// TwinCAT 3 PLC project PLCSim
// ProgramVersion: 3.1.4022.3
// libraries:
//   Tc2_Standard, * (Beckhoff Automation GmbH)
//   Tc2_System, * (Beckhoff Automation GmbH)
//   Tc3_Module, * (Beckhoff Automation GmbH)
//   VisuSymbols,3.5.10.0,System
// project tree:
//   / GlobalTextList.TcGTLO, PlcTask.TcTTO (not stored), Visualization Manager.TcVMO (not stored)
//   POUs/ MAIN.TcPOU
//   VISUs/ Visualization.TcVIS

// ---- POUs/MAIN.TcPOU
PROGRAM MAIN
VAR
	ixLampStarted	AT %I* : BOOL;
	ixSliderAout 	AT %I* : BOOL; 
	ixSliderAin 	AT %I* : BOOL; 
	ixSliderBout 	AT %I* : BOOL; 
	ixSliderBin 	AT %I* : BOOL; 
	ixDrillDown 	AT %I* : BOOL;
	ixDrillUp		AT %I* : BOOL;
	
	qxButtonStart	AT %Q* : BOOL;
	qxButtonStop	AT %Q* : BOOL;
	qxSliderAout	AT %Q* : BOOL;
	qxSliderAin		AT %Q* : BOOL;
	qxSliderBout	AT %Q* : BOOL;
	qxSliderBin		AT %Q* : BOOL;
	qxDrillUp		AT %Q* : BOOL;
	qxDrillDown		AT %Q* : BOOL;
	
	mxReset 		: BOOL;
	mxCubeInvisible : BOOL;
	
	
	nPosSliderA 	: INT:=0;
	nPosSliderB 	: INT:=0;
	nPosDrill 		: INT:=0;
	nPosXCube		: INT:=0;
	nPosYCube		: INT:=0;
	nSpeed 			: INT:=1;
	nCnt			: INT:=0;
	nErrorCnt		: INT:=0;
	nSeq: INT;
	
	fbTONAin:TON;
	fbTONAout:TON;
	fbTONBin:TON;
	fbTONBout:TON;
	fbTONDrillUp:TON;
	fbTONADrillDown:TON;
	
	
END_VAR

// Anders Nilsson Exam 2022

// Slider A
IF ixSliderAout AND NOT ixSliderAin THEN
	nPosSliderA := nPosSliderA-nSpeed;
	IF nPosSliderA < -75 THEN
		nPosSliderA := -75;
	END_IF
END_IF

IF ixSliderAin AND NOT ixSliderAout THEN
	nPosSliderA := nPosSliderA+nSpeed;
	IF nPosSliderA > 0 THEN
		nPosSliderA := 0;
	END_IF
END_IF

fbTONAin.PT := T#1S;
fbTONAin.IN := nPosSliderA = 0;
fbTONAin();
qxSliderAin := fbTONAin.Q;

fbTONAout.PT := T#1S;
fbTONAout.IN := nPosSliderA = -75;
fbTONAout();
qxSliderAout := fbTONAout.Q;



// Slider B
IF ixSliderBout AND NOT ixSliderBin THEN
	nPosSliderB := nPosSliderB + nSpeed;
	IF nPosSliderB > 0 THEN
		nPosSliderB := 0;
	END_IF
	
END_IF

IF ixSliderBin AND NOT ixSliderBout THEN
	nPosSliderB := nPosSliderB - nSpeed;
	IF nPosSliderB< -75 THEN
		nPosSliderB := -75;
	END_IF
END_IF

fbTONBin.PT := T#1S;
fbTONBin.IN := nPosSliderB = -75;
fbTONBin();
qxSliderBin := fbTONBin.Q;

fbTONBout.PT := T#1S;
fbTONBout.IN := nPosSliderB = 0;
fbTONBout();
qxSliderBout := fbTONBout.Q;




// Drill 
IF ixDrillDown AND NOT ixDrillUp THEN
	nPosDrill := nPosDrill + nSpeed;
	IF nPosDrill > 35 THEN
		nPosDrill := 35;
	END_IF
END_IF
	
IF ixDrillUp AND NOT ixDrillDown THEN
	nPosDrill := nPosDrill - nSpeed;
	IF nPosDrill < 0 THEN
		nPosDrill := 0;
	END_IF
END_IF
	
fbTONDrillUp.PT := T#1S;
fbTONDrillUp.IN := nPosDrill = 0;
fbTONDrillUp();
qxDrillUp := fbTONDrillUp.Q;

fbTONADrillDown.PT := T#1S;
fbTONADrillDown.IN := nPosDrill = 35;
fbTONADrillDown();
qxDrillDown := fbTONADrillDown.Q;


	
IF	mxReset THEN
	nSeq 		:= 10;
	nCnt 		:= 0;
	nErrorCnt   := 0;
	nPosSliderA := 0;
	nPosSliderB := 0;
	nPosDrill 	:= 0;
	nPosXCube   := 0;
	nPosYCube   := 0;
	mxCubeInvisible := FALSE;
END_IF
	

	
// Cube
CASE nSeq OF 
	0: 	//Start and Init Slider A in position
		IF 	qxSliderAIn THEN
			nPosXCube := 0;
		    nPosYCube := 0;
			mxCubeInvisible := FALSE;
			nSeq := 10;
		END_IF
		
	10:	//Slide A out
		nPosXCube := nPosSliderA;
		IF qxSliderAout THEN
			nSeq := 20;
		END_IF
		
		//Error
		IF  ixSliderAout AND ( NOT qxSliderBout OR NOT qxDrillUp) THEN
			nSeq := 100;
		END_IF
	
		
	20:	//Drill
	
		IF qxDrillDown THEN
			nSeq := 30;
		END_IF
		
		//Error
		IF 	NOT qxSliderAout OR NOT qxSliderBout  THEN
			nSeq := 100;
		END_IF
		
		
	30:  //Slide B in cube out
	
	    IF qxSliderBin AND NOT qxSliderAout THEN
			nCnt := nCnt +1;
			mxCubeInvisible := TRUE;
			nSeq := 0;
		END_IF
			
	100: //Error
		mxCubeInvisible := TRUE;
		IF 	qxSliderAIn THEN
			nErrorCnt := nErrorCnt +1;
			nSeq := 0;
		END_IF
	
	
END_CASE

END_PROGRAM

// ---- GlobalTextList.TcGTLO
TEXTLIST GlobalTextList
  372 = 'A'
  923 = 'B'
  661 = 'Counter'
  201 = 'Counter %S'
  776 = 'Counter %s'
  882 = 'Counter %sCounter %s'
  36 = 'Cylibder B'
  529 = 'Cylibders B'
  223 = 'Cylinder A'
  735 = 'Cylinder B'
  726 = 'Drill'
  832 = 'Drill Plant'
  634 = 'Errors %s'
  926 = 'In'
  848 = 'Manover'
  431 = 'Nilsson'
  255 = 'Nilsson\nzz'
  607 = 'Out'
  719 = 'Pusher'
  311 = 'Reset'
  761 = 'Slider A'
  571 = 'Slider B'
  532 = 'Start'
  630 = 'Stop'
  348 = 'University West'
  517 = 'University West\nAnders Nilsson'
  245 = 'University West\nAnders Nilsson Nov 2019'
  193 = 'University West\nAnders Nilsson Nov 2022'
END_TEXTLIST

// ---- VISUs/Visualization.TcVIS
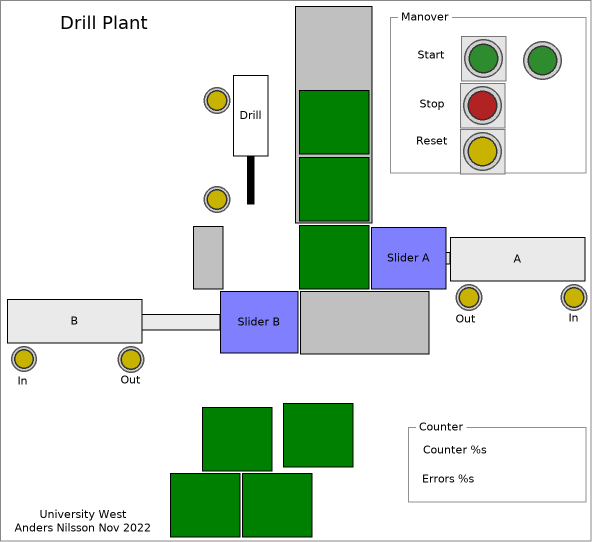
VISUALIZATION Visualization  // 592x542
    Group (233,75 59x138)
        p2773130477: main.nPosDrill
        p1126004900: MAIN.nPosDrill
        Rectangle (0,0 35x81), "Drill"
        Rectangle (14,81 7x48)
    Rectangle (295,6 77x217)
    Rectangle (299,225 70x64), invisible if: MAIN.mxCubeInvisible
        p3528305787: MAIN.nPosXCube
        p874137650: MAIN.nPosXCube
        p2773130477: MAIN.nPosYCube
        p1126004900: MAIN.nPosYCube
    Rectangle (193,226 30x63)
    Rectangle (299,157 70x64)
    Rectangle (300,291 129x63)
    Rectangle (299,90 70x64)
    Lamp1 (115,344 32x31), variable: MAIN.qxSliderBout, style: Lamp-Lamp1-Yellow
    Lamp1 (8,344 32x30), variable: MAIN.qxSliderBin, style: Lamp-Lamp1-Yellow
    Lamp1 (558,282 32x31), variable: MAIN.qxSliderAin, style: Lamp-Lamp1-Yellow
    Lamp1 (453,282 32x31), variable: MAIN.qxSliderAout, style: Lamp-Lamp1-Yellow
    Lamp1 (201,85 32x31), variable: MAIN.qxDrillUp, style: Lamp-Lamp1-Yellow
    Lamp1 (201,184 32x31), variable: MAIN.qxDrillDown, style: Lamp-Lamp1-Yellow
    Rectangle (242,473 70x64), invisible if: main.nCnt < 1
    Rectangle (283,403 70x64), invisible if: main.nCnt < 4
    Rectangle (170,473 70x64), invisible if: main.nCnt < 2
    Rectangle (202,407 70x64), invisible if: main.nCnt < 3
    GroupBox (390,9 196x164), "Manover"
        Label (20,23 42x46), "Start"
        PushSwitch (71,27 45x45), variable: MAIN.qxButtonStart, behaviour: TAP, style: Switch-PushSwitch-Green
        PushSwitch (70,74 45x45), variable: MAIN.qxButtonStop, behaviour: TAP, style: Switch-PushSwitch-Red
        Lamp1 (130,29 45x45), variable: MAIN.ixLampStarted, style: Lamp-Lamp1-Green
        Label (21,72 42x46), "Stop"
        PushSwitch (70,120 45x45), variable: MAIN.mxReset, behaviour: TAP, style: Switch-PushSwitch-Yellow
    GroupBox (408,419 178x83), "Counter"
        Rectangle (12,16 112x30), "Counter %s", text variable: MAIN.nCnt
        Rectangle (11,45 112x30), "Errors %s", text variable: MAIN.nErrorCnt
    Label (447,302 37x34), "Out"
    Label (112,363 37x34), "Out"
    Label (555,301 37x34), "In"
    Label (4,364 37x34), "In"
    Label (411,118 42x46), "Reset"
    Rectangle (371,252 79x12)
    Rectangle (450,237 135x44), "A"
    Rectangle (139,314 81x16)
    Rectangle (7,299 135x44), "B"
    Rectangle (371,227 75x62), "Slider A"
        p3528305787: MAIN.nPosSliderA
        p874137650: MAIN.nPosSliderA
    Rectangle (220,291 78x62), "Slider B"
        p3528305787: MAIN.nPosSliderB
        p874137650: MAIN.nPosSliderB
    Label (26,6 156x34), "Drill Plant"
    Label (7,500 152x42), "University West Anders Nilsson Nov 2022"
END_VISUALIZATION
